Staubli VAL3: ioWrite.pgx

public program ioWrite(num& x_nMsgRecvState)
  local bool l_bOk
  local num l_nCounter
  local num l_nJointError
  local MotionCmd l_mTrajPt
begin
  // Copyright (c) 2016, Ocado Technology - Robotics Research Team
  //
  // Licensed under the Apache License, Version 2.0 (the "License");
  // you may not use this file except in compliance with the License.
  // You may obtain a copy of the License at
  //
  //     http://www.apache.org/licenses/LICENSE-2.0
  //
  // Unless required by applicable law or agreed to in writing, software
  // distributed under the License is distributed on an "AS IS" BASIS,
  // WITHOUT WARRANTIES OR CONDITIONS OF ANY KIND, either express or implied.
  // See the License for the specific language governing permissions and
  // limitations under the License.


  logMsg("IOWRITE"+toString("", rosIoWriteRequestMsg.ioWriteRequest.nIndex))

  tTool.gripper = false
  delay(2)
  tTool.gripper = true
  delay(2)
    tTool.gripper = false
  delay(2)
  tTool.gripper = true
  delay(2)
    tTool.gripper = false
  delay(2)
  tTool.gripper = true
  delay(2)

  //if (rosIoWriteRequestMsg.ioWriteRequest.nIndex == 1)
    if (rosIoWriteRequestMsg.ioWriteRequest.nValue==0)
       tTool.gripper = false
    else
       tTool.gripper = true
    endIf
  //endIf


    if (l_bOk==false)
      // could not push trajectory point into buffer
      // thus ACK should flag FAILURE, but only if comm type is request
      if (rosGenericMsg.header.nCommType==2)

            rosIoWriteRequestAck.header.nReplyCode=2

      endIf
    endIf

  // check whether ACK should be sent
  if (rosGenericMsg.header.nCommType == 2)
    // comm type request requires ACK
    x_nMsgRecvState = 5
  else
    // other comm types (e.g., topic) does not require ACK, hence skip state
    x_nMsgRecvState = 0
  endIf
end
